// Asserts that two ULINTs are equal. If they are not, an assertion error is created.
METHOD PUBLIC AssertEquals_ULINT
VAR_INPUT
    Expected : ULINT; // ULINT expected value
    Actual : ULINT; // ULINT actual value
    Message : T_MaxString; // The identifying message for the assertion error
END_VAR
VAR
    TestInstancePath : T_MaxString;
    AlreadyReported : BOOL;
END_VAR
IF GVL_TcUnit.IgnoreCurrentTest OR GVL_TcUnit.CurrentTestIsFinished THEN
    RETURN;
END_IF

TestInstancePath := AddTestNameToInstancePath(TestInstancePath := FindTestSuiteInstancePath());

AssertResults.ReportResult(ExpectedSize := SIZEOF(Expected),
                           ExpectedTypeClass := IBaseLibrary.TypeClass.TYPE_ULINT,
                           ExpectedValue := ADR(Expected),
                           ActualSize := SIZEOF(Actual),
                           ActualTypeClass := IBaseLibrary.TypeClass.TYPE_ULINT,
                           ActualValue := ADR(Actual),
                           Message := Message,
                           TestInstancePath := TestInstancePath,
                           AlreadyReported => AlreadyReported);

IF NOT AlreadyReported AND Expected <> Actual THEN
    SetTestFailed(AssertionType := E_AssertionType.Type_ULINT,
                  AssertionMessage := Message);

    AssertMessageFormatter.LogAssertFailure(Expected := ULINT_TO_STRING(Expected),
                                            Actual := ULINT_TO_STRING(Actual),
                                            Message := Message,
                                            TestInstancePath := TestInstancePath);
END_IF
END_METHOD

// Asserts that two USINTs are equal. If they are not, an assertion error is created.
METHOD PUBLIC AssertEquals_USINT
VAR_INPUT
    Expected : USINT; // USINT expected value
    Actual : USINT; // USINT actual value
    Message : T_MaxString; // The identifying message for the assertion error
END_VAR
VAR
    AlreadyReported : BOOL;
    TestInstancePath : T_MaxString;
END_VAR
IF GVL_TcUnit.IgnoreCurrentTest OR GVL_TcUnit.CurrentTestIsFinished THEN
    RETURN;
END_IF

TestInstancePath := AddTestNameToInstancePath(TestInstancePath := FindTestSuiteInstancePath());

AssertResults.ReportResult(ExpectedSize := SIZEOF(Expected),
                           ExpectedTypeClass := IBaseLibrary.TypeClass.TYPE_USINT,
                           ExpectedValue := ADR(Expected),
                           ActualSize := SIZEOF(Actual),
                           ActualTypeClass := IBaseLibrary.TypeClass.TYPE_USINT,
                           ActualValue := ADR(Actual),
                           Message := Message,
                           TestInstancePath := TestInstancePath,
                           AlreadyReported => AlreadyReported);

IF NOT AlreadyReported AND Expected <> Actual THEN
    SetTestFailed(AssertionType := E_AssertionType.Type_USINT,
                  AssertionMessage := Message);

    AssertMessageFormatter.LogAssertFailure(Expected := USINT_TO_STRING(Expected),
                                            Actual := USINT_TO_STRING(Actual),
                                            Message := Message,
                                            TestInstancePath := TestInstancePath);
END_IF
END_METHOD

// Asserts that two WORDs are equal. If they are not, an assertion error is created.
METHOD PUBLIC AssertEquals_WORD
VAR_INPUT
    Expected : WORD; // WORD expected value
    Actual : WORD; // WORD actual value
    Message : T_MaxString; // The identifying message for the assertion error
END_VAR
VAR
    TestInstancePath : T_MaxString;
    AlreadyReported : BOOL;
END_VAR
IF GVL_TcUnit.IgnoreCurrentTest OR GVL_TcUnit.CurrentTestIsFinished THEN
    RETURN;
END_IF

TestInstancePath := AddTestNameToInstancePath(TestInstancePath := FindTestSuiteInstancePath());

AssertResults.ReportResult(ExpectedSize := SIZEOF(Expected),
                           ExpectedTypeClass := IBaseLibrary.TypeClass.TYPE_WORD,
                           ExpectedValue := ADR(Expected),
                           ActualSize := SIZEOF(Actual),
                           ActualTypeClass := IBaseLibrary.TypeClass.TYPE_WORD,
                           ActualValue := ADR(Actual),
                           Message := Message,
                           TestInstancePath := TestInstancePath,
                           AlreadyReported => AlreadyReported);

IF NOT AlreadyReported AND Expected <> Actual THEN
    SetTestFailed(AssertionType := E_AssertionType.Type_WORD,
                  AssertionMessage := Message);

    AssertMessageFormatter.LogAssertFailure(Expected := CONCAT(
                                                            STR1 := '0x',
                                                            STR2 := WORD_TO_HEXSTR(in := Expected,
                                                                                                 iPrecision := 4,
                                                                                                 bLoCase := FALSE)),
                                            Actual := CONCAT(
                                                            STR1 := '0x',
                                                            STR2 := WORD_TO_HEXSTR(in := Actual,
                                                                                                 iPrecision := 4,
                                                                                                 bLoCase := FALSE)),
                                            Message := Message,
                                            TestInstancePath := TestInstancePath);
END_IF
END_METHOD

// Asserts that two WSTRINGs are equal. If they are not, an assertion error is created.
METHOD PUBLIC AssertEquals_WSTRING
VAR_INPUT
    Expected : WSTRING(255); // WSTRING expected value
    Actual : WSTRING(255); // WSTRING actual value
    Message : T_MaxString; // The identifying message for the assertion error
END_VAR
VAR
    TestInstancePath : T_MaxString;
    AlreadyReported : BOOL;
END_VAR
IF GVL_TcUnit.IgnoreCurrentTest OR GVL_TcUnit.CurrentTestIsFinished THEN
    RETURN;
END_IF

TestInstancePath := AddTestNameToInstancePath(TestInstancePath := FindTestSuiteInstancePath());

AssertResults.ReportResult(ExpectedSize := SIZEOF(Expected),
                           ExpectedTypeClass := IBaseLibrary.TypeClass.TYPE_WSTRING,
                           ExpectedValue := ADR(Expected),
                           ActualSize := SIZEOF(Actual),
                           ActualTypeClass := IBaseLibrary.TypeClass.TYPE_WSTRING,
                           ActualValue := ADR(Actual),
                           Message := Message,
                           TestInstancePath := TestInstancePath,
                           AlreadyReported => AlreadyReported);

IF NOT AlreadyReported AND (WLEN(STR := Expected) <> WLEN(STR := Actual) OR (Expected <> Actual)) THEN
    SetTestFailed(AssertionType := E_AssertionType.Type_WSTRING,
                  AssertionMessage := Message);

    AssertMessageFormatter.LogAssertFailure(Expected := 'Not possible to print EXP unicode WSTRING value',
                                            Actual := 'Not possible to print ACT unicode WSTRING value',
                                            Message := Message,
                                            TestInstancePath := TestInstancePath);
END_IF
END_METHOD

// Asserts that a condition is false. If it is not, an assertion error is created.
METHOD PUBLIC AssertFalse
VAR_INPUT
    Condition : BOOL; // Condition to be checked
    Message : T_MaxString; // The identifying message for the assertion error
END_VAR
AssertEquals_BOOL(Expected := FALSE,
                  Actual := Condition,
                  Message := Message);
END_METHOD

// Asserts that a condition is true. If it is not, an assertion error is created.
METHOD PUBLIC AssertTrue
VAR_INPUT
    Condition : BOOL; // Condition to be checked
    Message : T_MaxString; // The identifying message for the assertion error
END_VAR
AssertEquals_BOOL(Expected := TRUE,
                  Actual := Condition,
                  Message := Message);
END_METHOD

METHOD INTERNAL CalculateAndSetNumberOfAssertsForTest
VAR_INPUT
    TestName : T_MaxString;
END_VAR
VAR
    TestInstancePath : T_MaxString;
    TotalNumberOfAsserts : UINT;
    NumberOfAsserts : UINT;
    NumberOfArrayAsserts : UINT;
    
    IteratorCounter : UINT;
END_VAR
TestInstancePath := AddTestNameToInstancePath(FindTestSuiteInstancePath());
NumberOfAsserts := AssertResults.GetNumberOfAssertsForTest(CompleteTestInstancePath := TestInstancePath);
NumberOfArrayAsserts := AssertArrayResults.GetNumberOfArrayAssertsForTest(CompleteTestInstancePath := TestInstancePath);
TotalNumberOfAsserts := NumberOfAsserts + NumberOfArrayAsserts;

IF TotalNumberOfAsserts > 0 THEN
    IF NumberOfTests > 0 THEN
        FOR IteratorCounter := 1 TO NumberOfTests BY 1 DO
            IF Tests[IteratorCounter].GetName() = TestName THEN
                Tests[IteratorCounter].SetNumberOfAssertions(NoOfAssertions := TotalNumberOfAsserts);
                RETURN;
            END_IF
        END_FOR
    END_IF
END_IF
END_METHOD

METHOD INTERNAL CalculateDuration
VAR_INPUT
    FinishedAt : LWORD; // CPU cycle counter with 100ns precision
END_VAR
IF Duration = 0.0 THEN
	Duration := LWORD_TO_LREAL(FinishedAt - StartedAt) * GVL_TcUnit.HundredNanosecondToSecond; // Seconds
	TraceWithSeverity(
		Message := CONCAT(CONCAT('SUITE COMPLETE: ', InstancePath),
				   CONCAT(' - ', CONCAT(UINT_TO_STRING(GetNumberOfSuccessfulTests()), CONCAT(' passed, ',
				   CONCAT(UINT_TO_STRING(GetNumberOfFailedTests()), CONCAT(' failed, ',
				   CONCAT(UINT_TO_STRING(GetNumberOfSkippedTests()), CONCAT(' skipped (',
				   CONCAT(LREAL_TO_STRING(Duration), 's)'))))))))),
		Severity := Global.TcEventSeverity.Info);
END_IF
END_METHOD

METHOD FB_init : BOOL
VAR_INPUT
    bInitRetains : BOOL; // if TRUE, the retain variables are initialized (warm start / cold start)
    bInCopyCode : BOOL;  // if TRUE, the instance afterwards gets moved into the copy code (online change)
END_VAR
GVL_TcUnit.NumberOfInitializedTestSuites := GVL_TcUnit.NumberOfInitializedTestSuites + 1;
GVL_TcUnit.TestSuiteAddresses[GVL_TcUnit.NumberOfInitializedTestSuites] := THIS;
END_METHOD

// Searches for the instance path of the calling function block
METHOD PRIVATE FindTestSuiteInstancePath : T_MaxString
FindTestSuiteInstancePath := GetInstancePath();
END_METHOD

METHOD INTERNAL GetDuration : LREAL
GetDuration := Duration;
END_METHOD

METHOD INTERNAL GetHasStartedRunning : BOOL
GetHasStartedRunning := StartedAt > 0;
END_METHOD

METHOD INTERNAL GetInstancePath : T_MaxString
GetInstancePath := InstancePath;
END_METHOD

METHOD INTERNAL GetNumberOfFailedTests : UINT
VAR
    Counter : UINT;
    FailedTestsCount : UINT;
    NumberOfTestsToAnalyse : UINT(1..GVL_Param_TcUnit.MaxNumberOfTestsForEachTestSuite);
    NumberOfTestOverArrayLimit : UINT;
END_VAR
// Limit the test analyse to the max array limit of 'Tests[]'
NumberOfTestsToAnalyse := GetNumberOfTestsToAnalyse();
IF GetNumberOfTests() > NumberOfTestsToAnalyse THEN
    NumberOfTestOverArrayLimit := GetNumberOfTests()-NumberOfTestsToAnalyse;
END_IF

FOR Counter := 1 TO NumberOfTestsToAnalyse BY 1 DO
    IF Tests[Counter].IsFailed() THEN
        FailedTestsCount := FailedTestsCount + 1;
    END_IF
END_FOR

GetNumberOfFailedTests := FailedTestsCount + NumberOfTestOverArrayLimit;
END_METHOD

METHOD INTERNAL GetNumberOfSkippedTests : UINT
VAR
    Counter : UINT;
    SkippedTestsCount : UINT;
    NumberOfTestsToAnalyse : UINT(1..GVL_Param_TcUnit.MaxNumberOfTestsForEachTestSuite);
END_VAR
// Limit the test analyse to the max array limit of 'Tests[]'
NumberOfTestsToAnalyse := GetNumberOfTestsToAnalyse();

FOR Counter := 1 TO NumberOfTestsToAnalyse BY 1 DO
    IF Tests[Counter].IsSkipped() THEN
        SkippedTestsCount := SkippedTestsCount + 1;
    END_IF
END_FOR

GetNumberOfSkippedTests := SkippedTestsCount;
END_METHOD

METHOD INTERNAL GetNumberOfSuccessfulTests : UINT
GetNumberOfSuccessfulTests := GetNumberOfTests() - GetNumberOfFailedTests() - GetNumberOfSkippedTests();
END_METHOD

METHOD INTERNAL GetNumberOfTests : UINT
GetNumberOfTests := NumberOfTests;
END_METHOD

METHOD INTERNAL GetNumberOfTestsToAnalyse : UINT
GetNumberOfTestsToAnalyse := MIN(GetNumberOfTests(), GVL_Param_TcUnit.MaxNumberOfTestsForEachTestSuite);
END_METHOD

METHOD GetTestByName : REFERENCE TO FB_Test
VAR_INPUT
  TestName : T_MaxString;
END_VAR
VAR
  IteratorCounter : UINT;
  NumberOfTestsToAnalyse : UINT(1..GVL_Param_TcUnit.MaxNumberOfTestSuites);
END_VAR
NumberOfTestsToAnalyse := GetNumberOfTestsToAnalyse();
FOR IteratorCounter := 1 TO NumberOfTestsToAnalyse BY 1 DO
  IF Tests[IteratorCounter].GetName() = TestName THEN
    GetTestByName REF= Tests[IteratorCounter];
    RETURN;
	END_IF
END_FOR
END_METHOD

// This method returns the test at the n'th position, ranging from 1.. NumberOfTests
METHOD INTERNAL GetTestByPosition : FB_Test
VAR_INPUT
    Position : UINT(1..GVL_Param_TcUnit.MaxNumberOfTestsForEachTestSuite);
END_VAR
GetTestByPosition := Tests[Position];
END_METHOD

METHOD INTERNAL GetTestOrderNumber : UINT(0..GVL_Param_TcUnit.MaxNumberOfTestsForEachTestSuite);
VAR_INPUT
    TestName : T_MaxString;
END_VAR
VAR
    IteratorCounter : UINT;
    NumberOfTestsToAnalyse : UINT(1..GVL_Param_TcUnit.MaxNumberOfTestsForEachTestSuite);
END_VAR
// Limit the test analyse to the max array limit of 'Tests[]'
NumberOfTestsToAnalyse := GetNumberOfTestsToAnalyse();

FOR IteratorCounter := 1 TO NumberOfTestsToAnalyse BY 1 DO
    IF Tests[IteratorCounter].GetName() = TestName THEN
        GetTestOrderNumber := Tests[IteratorCounter].GetTestOrder();
        RETURN;
    END_IF
END_FOR
END_METHOD

METHOD INTERNAL IsTestFinished : BOOL
VAR_INPUT
    TestName : T_MaxString;
END_VAR
VAR
    IteratorCounter : UINT;
    NumberOfTestsToAnalyse : UINT(0..GVL_Param_TcUnit.MaxNumberOfTestsForEachTestSuite);
END_VAR
// Limit the test analyse to the max array limit of 'Tests[]'
NumberOfTestsToAnalyse := GetNumberOfTestsToAnalyse();

IsTestFinished := FALSE;
FOR IteratorCounter := 1 TO NumberOfTestsToAnalyse BY 1 DO
    IF Tests[IteratorCounter].GetName() = TestName THEN
        IsTestFinished := Tests[IteratorCounter].IsFinished();
        RETURN;
    END_IF
END_FOR
END_METHOD

METHOD INTERNAL SetStartedAtIfNotSet
VAR_INPUT
    Timestamp : LWORD; // CPU cycle counter with 100ns precision
END_VAR
IF StartedAt = 0 THEN
    StartedAt := Timestamp;
END_IF
END_METHOD

METHOD INTERNAL SetStartedAtTimeBasedOnCpuCounter
StartedAt := F_GetCpuCounterAs64bit(GVL_TcUnit.GetCpuCounter);
END_METHOD

METHOD INTERNAL SetTestFailed
VAR_INPUT
    AssertionType : E_AssertionType;
    AssertionMessage : T_MaxString;
END_VAR
VAR
    IteratorCounter : UINT;
    NumberOfTestsToAnalyse : UINT(0..GVL_Param_TcUnit.MaxNumberOfTestsForEachTestSuite);
END_VAR
// Limit the test analyse to the max array limit of 'Tests[]'
NumberOfTestsToAnalyse := GetNumberOfTestsToAnalyse();

FOR IteratorCounter := 1 TO NumberOfTestsToAnalyse BY 1 DO
    IF Tests[IteratorCounter].GetName() = GVL_TcUnit.CurrentTestNameBeingCalled THEN
        Tests[IteratorCounter].SetFailed();
        Tests[IteratorCounter].SetAssertionType(AssertType := AssertionType);
        Tests[IteratorCounter].SetAssertionMessage(AssertMessage := AssertionMessage);
    END_IF
END_FOR
END_METHOD

(* Marks the test as finished in this testsuite.
   Returns TRUE if test was found, and FALSE if a test with this name was not found in this testsuite *)
METHOD INTERNAL SetTestFinished : BOOL;
VAR_INPUT
    TestName : T_MaxString;
    FinishedAt : LWORD;
END_VAR
VAR
    IteratorCounter : UINT;
    NumberOfTestsToAnalyse : UINT(0..GVL_Param_TcUnit.MaxNumberOfTestsForEachTestSuite);
END_VAR
// Limit the test analyse to the max array limit of 'Tests[]'
NumberOfTestsToAnalyse := GetNumberOfTestsToAnalyse();
FOR IteratorCounter := 1 TO NumberOfTestsToAnalyse BY 1 DO
    IF Tests[IteratorCounter].GetName() = TestName THEN
		IF NOT Tests[IteratorCounter].IsFinished() THEN
        	Tests[IteratorCounter].SetFinishedAndDuration(FinishedAt := FinishedAt);
			IF Tests[IteratorCounter].IsFailed() THEN
				TraceWithSeverity(
					Message := CONCAT(CONCAT('TEST FAILED: ', TestName),
							   CONCAT(' (', CONCAT(LREAL_TO_STRING(Tests[IteratorCounter].GetDuration()), 's)'))),
					Severity := Global.TcEventSeverity.Warning);
			ELSE
				TraceWithSeverity(
					Message := CONCAT(CONCAT('TEST PASSED: ', TestName),
							   CONCAT(' (', CONCAT(LREAL_TO_STRING(Tests[IteratorCounter].GetDuration()), 's)'))),
					Severity := Global.TcEventSeverity.Info);
			END_IF
		END_IF
		SetTestFinished := TRUE;
        RETURN;
    END_IF
END_FOR
SetTestFinished := FALSE;
END_METHOD

END_FUNCTION_BLOCK

// POUs/FB_xUnitXmlPublisher
// Publishes test results into an xUnit compatible Xml file
FUNCTION_BLOCK FB_xUnitXmlPublisher EXTENDS FB_BaseStatic IMPLEMENTS I_TestResultLogger
VAR
    // Dependency injection via FB_Init
    TestResults : I_TestResults;

    // File access mode
    AccessMode : SysFile.ACCESS_MODE := SysFile.AM_WRITE_PLUS;

    File : FB_FileControl;
    Xml : FB_XMLControl;
    BufferInitialised : BOOL := FALSE;
    Buffer : ARRAY [0..(GVL_Param_TcUnit.XUnitBufferSize - 1)] OF BYTE;
    WritingTestSuiteResultNumber : UINT(1..GVL_Param_TcUnit.MaxNumberOfTestSuites);
    PublishTrigger : R_TRIG;
END_VAR

(*
    Deletes the former file (if it exists).
    Opens the file, writes the buffer and closes it.
*)
METHOD PRIVATE DeleteOpenWriteClose : SysFile.SysTypes.RTS_IEC_RESULT;
VAR
    WriteResult : SysFile.SysTypes.RTS_IEC_RESULT;
END_VAR
DeleteOpenWriteClose := SysDir.CmpErrors.Errors.ERR_OK;
IF Initialised() THEN
    // Delete may fail if file doesn't exist yet (first run) — not a real error
    DeleteOpenWriteClose := MAX(DeleteOpenWriteClose, File.Delete(Filename := GVL_Param_TcUnit.xUnitFilePath));
    // Track Open/Write/Close separately for trace — these are the real errors
    WriteResult := File.Open(Filename := GVL_Param_TcUnit.xUnitFilePath, FileAccessMode := AccessMode);
    WriteResult := MAX(WriteResult, File.Write(BufferPointer := ADR(Buffer), Xml.Length));
    WriteResult := MAX(WriteResult, File.Close());
    DeleteOpenWriteClose := MAX(DeleteOpenWriteClose, WriteResult);
ELSE
    WriteResult := SysDir.CmpErrors.Errors.ERR_NOBUFFER;
    DeleteOpenWriteClose := WriteResult;
END_IF;

IF WriteResult <> SysDir.CmpErrors.Errors.ERR_OK THEN
    TraceWithSeverity(
        Message := CONCAT('xUnit file I/O failure: ', GVL_Param_TcUnit.xUnitFilePath),
        Severity := Global.TcEventSeverity.Error);
END_IF;
END_METHOD

(*
    FB_Init is always available implicitly AND it is used primarily FOR initialization.
    The return value is not evaluated. For a specific influence, you can also declare the
    methods explicitly and provide additional code there with the standard initialization
    code. You can evaluate the return value.
*)
METHOD FB_Init: BOOL
VAR_INPUT
    bInitRetains: BOOL; // TRUE: the retain variables are initialized (reset warm / reset cold)
    bInCopyCode: BOOL;  // TRUE: the instance will be copied to the copy code afterward (online change)
    iTestResults : I_TestResults; // Interface dependency injection
END_VAR
// Set buffer and flag
Xml.SetBuffer(PointerToBuffer := ADR(Buffer), SizeOfBuffer := SIZEOF(Buffer));

// Set buffer initialised
BufferInitialised := TRUE;

// Set testresult interface
THIS^.TestResults := iTestResults;
END_METHOD

METHOD PRIVATE Initialised : BOOL
Initialised := THIS^.BufferInitialised;
END_METHOD

(*
    This method is responsible for the entire generation of the output file. 
    The output of the xml writer is NOT beautified.

    When new data is available, feel free to add it to the report
*)
METHOD PUBLIC LogTestSuiteResults
VAR
    UnitTestResults : REFERENCE TO ST_TestSuiteResults;
    CurrentSuiteNumber : UINT;
    CurrentTestCount : UINT;
END_VAR
VAR CONSTANT
    TEST_STATUS_SKIP : STRING := 'SKIP';
    TEST_STATUS_PASS : STRING := 'PASS';
    TEST_STATUS_FAIL : STRING := 'FAIL';
END_VAR
UnitTestResults REF= TestResults.GetTestSuiteResults();

// Only publish once if "GVL_Param_TcUnit.xUnitEnablePublish" is enabled and all test results are stored.
PublishTrigger(CLK := (TestResults.GetAreTestResultsAvailable() AND GVL_Param_TcUnit.xUnitEnablePublish));
IF PublishTrigger.Q THEN

    // <?xml version="1.0" encoding="UTF-8"?>
    Xml.WriteDocumentHeader(Header := '<?xml version="1.0" encoding="UTF-8"?>');

    // <testsuites>  ('disabled' removed 2026-07-18: an empty string breaks JUnit
    //  parsers expecting an integer; skipped counts carry the information)
    Xml.NewTag('testsuites');
    Xml.NewParameter('failures', UDINT_TO_STRING(UnitTestResults.NumberOfFailedTestCases));
    (* 'tests' is the TOTAL testcase count; the previous successful-only value was a bug *)
    Xml.NewParameter('tests', UDINT_TO_STRING(UnitTestResults.NumberOfTestCases));
    Xml.NewParameter('skipped', UDINT_TO_STRING(UnitTestResults.NumberOfSkippedTestCases));
    Xml.NewParameter('time', LREAL_TO_STRING(UnitTestResults.Duration));

    FOR CurrentSuiteNumber := 1 TO UnitTestResults.NumberOfTestSuites BY 1 DO
        // <testsuite>
        Xml.NewTag('testsuite');
        Xml.NewParameter('id', UINT_TO_STRING(UnitTestResults.TestSuiteResults[CurrentSuiteNumber].Identity));
        Xml.NewParameter('name', UnitTestResults.TestSuiteResults[CurrentSuiteNumber].name);
        Xml.NewParameter('tests', UINT_TO_STRING(UnitTestResults.TestSuiteResults[CurrentSuiteNumber].NumberOfTests));
        Xml.NewParameter('failures', UINT_TO_STRING(UnitTestResults.TestSuiteResults[CurrentSuiteNumber].NumberOfFailedTests));
        Xml.NewParameter('skipped', UINT_TO_STRING(UnitTestResults.TestSuiteResults[CurrentSuiteNumber].NumberOfSkippedTests));
        Xml.NewParameter('time', LREAL_TO_STRING(UnitTestResults.TestSuiteResults[CurrentSuiteNumber].Duration));

        FOR CurrentTestCount := 1 TO UnitTestResults.TestSuiteResults[CurrentSuiteNumber].NumberOfTests BY 1 DO
            // <testcase>
            Xml.NewTag('testcase');
            Xml.NewParameter('name', UnitTestResults.TestSuiteResults[CurrentSuiteNumber].TestCaseResults[CurrentTestCount].TestName);
            Xml.NewParameter('classname', UnitTestResults.TestSuiteResults[CurrentSuiteNumber].TestCaseResults[CurrentTestCount].TestClassName);
            Xml.NewParameter('time', LREAL_TO_STRING(UnitTestResults.TestSuiteResults[CurrentSuiteNumber].TestCaseResults[CurrentTestCount].Duration));

            IF UnitTestResults.TestSuiteResults[CurrentSuiteNumber].TestCaseResults[CurrentTestCount].TestIsFailed THEN
                Xml.NewParameter('status', TEST_STATUS_FAIL);
            ELSIF UnitTestResults.TestSuiteResults[CurrentSuiteNumber].TestCaseResults[CurrentTestCount].TestIsSkipped THEN
                Xml.NewParameter('status', TEST_STATUS_SKIP);
            ELSE
                Xml.NewParameter('status', TEST_STATUS_PASS);
            END_IF

            // Determine testcase fail, skip, or success
            IF UnitTestResults.TestSuiteResults[CurrentSuiteNumber].TestCaseResults[CurrentTestCount].FailureType <> E_AssertionType.Type_UNDEFINED THEN
                (* In case of fail
                    <failure message="Values differ" type="BYTE" />
                *)
                Xml.NewTag('failure');
                Xml.NewParameter('message', UnitTestResults.TestSuiteResults[CurrentSuiteNumber].TestCaseResults[CurrentTestCount].FailureMessage);
                Xml.NewParameter('type', F_AssertionTypeToString(UnitTestResults.TestSuiteResults[CurrentSuiteNumber].TestCaseResults[CurrentTestCount].FailureType));
                // Close failure tag
                Xml.CloseTag();
            ELSIF UnitTestResults.TestSuiteResults[CurrentSuiteNumber].TestCaseResults[CurrentTestCount].TestIsSkipped THEN
                (* JUnit consumers recognize a skipped testcase through a <skipped/>
                   child element, not a custom status attribute (kept for
                   backward compatibility) *)
                Xml.NewTag('skipped');
                Xml.CloseTag();
            ELSE
            // In case of success
            Xml.NewTagData('');

            END_IF
            // Close testcase tag
            Xml.CloseTag();

        END_FOR
        // Close testsuite tag
        Xml.CloseTag();

    END_FOR
    // Close testsuites
    Xml.CloseTag();

    // Delete, open, save and close the file
    DeleteOpenWriteClose();

    // Clear the internal buffer
    Xml.ClearBuffer();

    // Inform user
    GVL_TcUnit.AdsMessageQueue.WriteLog(MsgCtrlMask := ADSLOG_MSGTYPE_HINT,
                                        msgFmtStr := '%s',
                                        strArg := '| ==========TEST RESULTS EXPORTED===========');

    GVL_TcUnit.AdsMessageQueue.WriteLog(MsgCtrlMask := ADSLOG_MSGTYPE_HINT,
                                        msgFmtStr :=  '| Location: %s ',
                                        strArg := GVL_Param_TcUnit.xUnitFilePath);

    GVL_TcUnit.AdsMessageQueue.WriteLog(MsgCtrlMask := ADSLOG_MSGTYPE_HINT,
                                        MsgFmtStr := '%s',
                                        StrArg := '| ======================================');

    TraceWithSeverity(
        Message := CONCAT('xUnit XML exported to ', GVL_Param_TcUnit.xUnitFilePath),
        Severity := Global.TcEventSeverity.Info);
END_IF
END_METHOD

END_FUNCTION_BLOCK

// POUs/FB_TimedTestSuite
FUNCTION_BLOCK FB_TimedTestSuite EXTENDS FB_TestSuite
VAR
    TimedTestStates      : ARRAY[1..GVL_Param_TcUnit.MaxNumberOfTestsForEachTestSuite] OF ST_TimedTestState;
    _nActiveTimedTestIdx : UINT;
    (* Task cycle in which _nActiveTimedTestIdx was set; a wait helper only accepts
       the context if it was set in the same cycle (guards cross-scan staleness) *)
    _nActiveTimedTestCycle : UDINT;
    // One-shot for the out-of-context wait Error trace (cyclic path - must not storm)
    bOutOfContextWaitTraced : BOOL;
END_VAR

METHOD PRIVATE _FindTestIndex : UINT
VAR_INPUT
    TestName : T_MaxString;
END_VAR
VAR
    i : UINT;
    nMax : UINT;
END_VAR
_FindTestIndex := 0;
nMax := GetNumberOfTestsToAnalyse();
FOR i := 1 TO nMax BY 1 DO
    IF Tests[i].GetName() = TestName THEN
        _FindTestIndex := i;
        RETURN;
    END_IF
END_FOR
END_METHOD

(* Returns the timed-test index for a wait-helper call, or 0 when the call is
   out of context. Valid context requires all three: an index was set, it was
   set in the current task cycle (TEST_TIMED* ran earlier in this scan and
   selected this test for body execution), and the framework's current test
   name still matches (defense against later TEST() calls in the same scan). *)
METHOD PRIVATE _GetActiveWaitContext : UINT
VAR
    idx : UINT;
END_VAR
_GetActiveWaitContext := 0;
idx := _nActiveTimedTestIdx;
IF idx = 0 THEN
    RETURN;
END_IF

GetCurrentTaskIndex();
IF _nActiveTimedTestCycle <> TwinCAT_SystemInfoVarList._TaskInfo[GetCurrentTaskIndex.index].CycleCount THEN
    RETURN;
END_IF

IF Tests[idx].GetName() <> GVL_TcUnit.CurrentTestNameBeingCalled THEN
    RETURN;
END_IF

_GetActiveWaitContext := idx;
END_METHOD

METHOD PUBLIC GetTimedTestResult : ST_TimedTestResult
VAR_INPUT
    TestName : T_MaxString;
END_VAR
VAR
    idx  : UINT;
    Test : REFERENCE TO FB_Test;
END_VAR
// Normalize the same way TEST(), TEST_ORDERED(), and TEST_TIMED() do
TestName := F_LTrim(in := F_RTrim(in := TestName));

idx := _FindTestIndex(TestName := TestName);
IF idx = 0 THEN
    RETURN;
END_IF

Test REF= Tests[idx];
IF NOT __ISVALIDREF(Test) THEN
    RETURN;
END_IF

GetTimedTestResult.TestName := Test.GetName();
GetTimedTestResult.bIsFailed := Test.IsFailed();
GetTimedTestResult.bIsSkipped := Test.IsSkipped();
GetTimedTestResult.bIsFinished := Test.IsFinished();
GetTimedTestResult.sFailureMessage := Test.GetAssertionMessage();
GetTimedTestResult.eFailureType := Test.GetAssertionType();
GetTimedTestResult.nNumberOfAsserts := Test.GetNumberOfAssertions();
GetTimedTestResult.lrDuration := Test.GetDuration();
GetTimedTestResult.stTimedState := TimedTestStates[idx];
END_METHOD

METHOD PUBLIC TEST_TIMED : BOOL
VAR_INPUT
    TestName       : T_MaxString;
    tSafetyTimeout : TIME;
END_VAR
VAR
    idx         : UINT;
    lrElapsed   : LREAL;
    lrTimeout   : LREAL;
    sMsg        : T_MaxString;
END_VAR
TEST_TIMED := FALSE;

// Step 1: Reset context
_nActiveTimedTestIdx := 0;

// Step 2: Trim name
TestName := F_LTrim(in := F_RTrim(in := TestName));

// Step 3: Register test via free function TEST()
TEST(TestName := TestName);

// Step 4: Check skip/ignore
IF GVL_TcUnit.IgnoreCurrentTest THEN
    RETURN;
END_IF

// Step 5: Find test index
idx := _FindTestIndex(TestName := TestName);
IF idx = 0 THEN
    RETURN;
END_IF

// Step 6: Check already finished
IF TimedTestStates[idx].bSafetyTimedOut OR IsTestFinished(TestName := TestName) THEN
    GVL_TcUnit.CurrentTestIsFinished := TRUE;
    RETURN;
END_IF

// Step 7: Initialize on first call
IF NOT TimedTestStates[idx].bInitialized THEN
    TimedTestStates[idx].nSafetyStartTime := F_GetCpuCounterAs64bit(GVL_TcUnit.GetCpuCounter);
    TimedTestStates[idx].tSafetyTimeout := tSafetyTimeout;
    TimedTestStates[idx].bInitialized := TRUE;
END_IF

// Step 8: Check safety timeout (compare against stored value)
lrElapsed := ULINT_TO_LREAL(F_GetCpuCounterAs64bit(GVL_TcUnit.GetCpuCounter) - TimedTestStates[idx].nSafetyStartTime)
             * GVL_TcUnit.HundredNanosecondToSecond;
lrTimeout := TIME_TO_LREAL(TimedTestStates[idx].tSafetyTimeout) / 1000.0;

IF lrElapsed > lrTimeout THEN
    sMsg := CONCAT('SAFETY TIMEOUT: Test "', CONCAT(TestName, CONCAT('" exceeded ', LREAL_TO_FMTSTR(lrTimeout, 1, TRUE))));
    sMsg := CONCAT(sMsg, 's');

    SetTestFailed(AssertionType := E_AssertionType.Type_TIMEOUT,
                  AssertionMessage := sMsg);
    SetTestFinished(TestName := TestName,
                    FinishedAt := F_GetCpuCounterAs64bit(GVL_TcUnit.GetCpuCounter));
    CalculateAndSetNumberOfAssertsForTest(TestName := TestName);

    TimedTestStates[idx].bSafetyTimedOut := TRUE;
    GVL_TcUnit.CurrentTestIsFinished := TRUE;

    TraceWithSeverity(Message := sMsg, Severity := TcEventSeverity.Warning);
    RETURN;
END_IF

// Step 9: Test body should execute - arm the wait context for this cycle only
_nActiveTimedTestIdx := idx;
GetCurrentTaskIndex();
_nActiveTimedTestCycle := TwinCAT_SystemInfoVarList._TaskInfo[GetCurrentTaskIndex.index].CycleCount;
TEST_TIMED := TRUE;
END_METHOD

METHOD PUBLIC TEST_TIMED_ORDERED : BOOL
VAR_INPUT
    TestName       : T_MaxString;
    tSafetyTimeout : TIME;
END_VAR
VAR
    CounterTestSuiteAddress : UINT;
    SuiteIndex              : UINT;
    Test                    : REFERENCE TO FB_Test;
    idx                     : UINT;
    lrElapsed               : LREAL;
    lrTimeout               : LREAL;
    sMsg                    : T_MaxString;
END_VAR
TEST_TIMED_ORDERED := FALSE;

// Step 1: Reset context
_nActiveTimedTestIdx := 0;

// Step 2: Trim name (matches TEST_ORDERED line 34)
TestName := F_LTrim(in := F_RTrim(in := TestName));

// Step 3: Set global test name (matches line 37)
GVL_TcUnit.CurrentTestNameBeingCalled := TestName;

// Step 4: Find suite in runner registry (matches lines 44-47)
SuiteIndex := 0;
FOR CounterTestSuiteAddress := 1 TO GVL_TcUnit.NumberOfInitializedTestSuites BY 1 DO
    IF GVL_TcUnit.TestSuiteAddresses[CounterTestSuiteAddress] = GVL_TcUnit.CurrentTestSuiteBeingCalled THEN
        SuiteIndex := CounterTestSuiteAddress;
        EXIT;
    END_IF
END_FOR
IF SuiteIndex = 0 THEN
    RETURN;
END_IF

// Step 5: Register as ordered test (matches line 48)
Test REF= GVL_TcUnit.TestSuiteAddresses[SuiteIndex]^.AddTest(TestName := TestName, IsTestOrdered := TRUE);

// Step 6: Set CurrentTestIsFinished (matches line 49)
GVL_TcUnit.CurrentTestIsFinished := GVL_TcUnit.TestSuiteAddresses[SuiteIndex]^.IsTestFinished(TestName := TestName);

// Step 7: Check skip/ignore (matches lines 76-78)
IF GVL_TcUnit.IgnoreCurrentTest THEN
    RETURN;
END_IF

// Step 8: Check ordered cursor (matches lines 55-74)
IF GetTestOrderNumber(TestName := TestName) = GVL_TcUnit.CurrentlyRunningOrderedTestInTestSuite[SuiteIndex] THEN
    IF GVL_TcUnit.CurrentTestIsFinished THEN
        // Already finished - advance cursor (matches lines 58-62)
        GVL_TcUnit.CurrentlyRunningOrderedTestInTestSuite[SuiteIndex] :=
            GVL_TcUnit.CurrentlyRunningOrderedTestInTestSuite[SuiteIndex] + 1;
        GVL_TcUnit.IgnoreCurrentTest := TRUE;
        RETURN;
    END_IF
ELSE
    // Not this test's turn (matches lines 70-73)
    GVL_TcUnit.IgnoreCurrentTest := TRUE;
    RETURN;
END_IF

// --- From here: this test's turn AND not finished. Add timed-test logic. ---

// Step 9: Find timed test index
idx := _FindTestIndex(TestName := TestName);
IF idx = 0 THEN
    RETURN;
END_IF

// Step 10: Check already timed out
IF TimedTestStates[idx].bSafetyTimedOut THEN
    GVL_TcUnit.CurrentTestIsFinished := TRUE;
    RETURN;
END_IF

// Step 11: Initialize on first call
IF NOT TimedTestStates[idx].bInitialized THEN
    TimedTestStates[idx].nSafetyStartTime := F_GetCpuCounterAs64bit(GVL_TcUnit.GetCpuCounter);
    TimedTestStates[idx].tSafetyTimeout := tSafetyTimeout;
    TimedTestStates[idx].bInitialized := TRUE;
END_IF

// Step 12: Check safety timeout (compare against stored value)
lrElapsed := ULINT_TO_LREAL(F_GetCpuCounterAs64bit(GVL_TcUnit.GetCpuCounter) - TimedTestStates[idx].nSafetyStartTime)
             * GVL_TcUnit.HundredNanosecondToSecond;
lrTimeout := TIME_TO_LREAL(TimedTestStates[idx].tSafetyTimeout) / 1000.0;

IF lrElapsed > lrTimeout THEN
    sMsg := CONCAT('SAFETY TIMEOUT: Test "', CONCAT(TestName, CONCAT('" exceeded ', LREAL_TO_FMTSTR(lrTimeout, 1, TRUE))));
    sMsg := CONCAT(sMsg, 's');

    SetTestFailed(AssertionType := E_AssertionType.Type_TIMEOUT,
                  AssertionMessage := sMsg);
    SetTestFinished(TestName := TestName,
                    FinishedAt := F_GetCpuCounterAs64bit(GVL_TcUnit.GetCpuCounter));
    CalculateAndSetNumberOfAssertsForTest(TestName := TestName);

    TimedTestStates[idx].bSafetyTimedOut := TRUE;
    GVL_TcUnit.CurrentTestIsFinished := TRUE;

    TraceWithSeverity(Message := sMsg, Severity := TcEventSeverity.Warning);
    RETURN;
END_IF

// Step 13: Set started timestamp (matches line 66)
IF __ISVALIDREF(Test) THEN
    Test.SetStartedAtIfNotSet(Timestamp := F_GetCpuCounterAs64bit(GVL_TcUnit.GetCpuCounter));
END_IF

// Step 14: Test body should execute - arm the wait context for this cycle only
_nActiveTimedTestIdx := idx;
GetCurrentTaskIndex();
_nActiveTimedTestCycle := TwinCAT_SystemInfoVarList._TaskInfo[GetCurrentTaskIndex.index].CycleCount;
TEST_TIMED_ORDERED := TRUE;
END_METHOD

METHOD PUBLIC WaitForCondition : BOOL
VAR_INPUT
    bCondition : BOOL;
    tTimeout   : TIME;
END_VAR
VAR
    idx       : UINT;
    lrElapsed : LREAL;
    lrTarget  : LREAL;
END_VAR
WaitForCondition := FALSE;
idx := _GetActiveWaitContext();

// Step 1: Context check (one-shot trace - this path is cyclic)
IF idx = 0 THEN
    IF NOT bOutOfContextWaitTraced THEN
        bOutOfContextWaitTraced := TRUE;
        TraceWithSeverity(
            Message := 'WaitForCondition called without active timed test context',
            Severity := TcEventSeverity.Error);
    END_IF
    RETURN;
END_IF

// Step 2: Pass-through if already complete
IF TimedTestStates[idx].bWaitComplete THEN
    WaitForCondition := TRUE;
    RETURN;
END_IF

// Step 3: Type mismatch check
IF TimedTestStates[idx].eWaitType = E_WaitType.Duration THEN
    SetTestFailed(AssertionType := E_AssertionType.Type_WAIT_MISUSE,
                  AssertionMessage := 'WaitForCondition called but WaitForTime already active');
    SetTestFinished(TestName := GVL_TcUnit.CurrentTestNameBeingCalled,
                    FinishedAt := F_GetCpuCounterAs64bit(GVL_TcUnit.GetCpuCounter));
    CalculateAndSetNumberOfAssertsForTest(TestName := GVL_TcUnit.CurrentTestNameBeingCalled);
    GVL_TcUnit.CurrentTestIsFinished := TRUE;
    RETURN;
END_IF

// Step 4: First call with condition already TRUE - immediate completion
IF bCondition AND TimedTestStates[idx].nWaitStartTime = 0 THEN
    TimedTestStates[idx].bWaitComplete := TRUE;
    TimedTestStates[idx].bConditionTimedOut := FALSE;
    TimedTestStates[idx].eWaitType := E_WaitType.Condition;
    TraceWithSeverity(
        Message := CONCAT('WaitForCondition: condition already TRUE for test "', CONCAT(GVL_TcUnit.CurrentTestNameBeingCalled, '"')),
        Severity := TcEventSeverity.Info);
    WaitForCondition := TRUE;
    RETURN;
END_IF

// Step 5: First call, condition not yet met - start wait
IF TimedTestStates[idx].nWaitStartTime = 0 THEN
    TimedTestStates[idx].eWaitType := E_WaitType.Condition;
    TimedTestStates[idx].tLatchedDuration := tTimeout;
    TimedTestStates[idx].nWaitStartTime := F_GetCpuCounterAs64bit(GVL_TcUnit.GetCpuCounter);
    TraceWithSeverity(
        Message := CONCAT('WaitForCondition started: timeout ', CONCAT(TIME_TO_STRING(tTimeout), CONCAT(' for test "', CONCAT(GVL_TcUnit.CurrentTestNameBeingCalled, '"')))),
        Severity := TcEventSeverity.Verbose);
    RETURN;
END_IF

// Step 6: Condition met during wait
IF bCondition THEN
    TimedTestStates[idx].bWaitComplete := TRUE;
    TimedTestStates[idx].bConditionTimedOut := FALSE;
    TraceWithSeverity(
        Message := CONCAT('WaitForCondition: condition met for test "', CONCAT(GVL_TcUnit.CurrentTestNameBeingCalled, '"')),
        Severity := TcEventSeverity.Info);
    WaitForCondition := TRUE;
    RETURN;
END_IF

// Step 7: Check timeout
lrElapsed := ULINT_TO_LREAL(F_GetCpuCounterAs64bit(GVL_TcUnit.GetCpuCounter) - TimedTestStates[idx].nWaitStartTime)
             * GVL_TcUnit.HundredNanosecondToSecond;
lrTarget := TIME_TO_LREAL(TimedTestStates[idx].tLatchedDuration) / 1000.0;

IF lrElapsed >= lrTarget THEN
    TimedTestStates[idx].bWaitComplete := TRUE;
    TimedTestStates[idx].bConditionTimedOut := TRUE;
    TraceWithSeverity(
        Message := CONCAT('WaitForCondition timed out after ', CONCAT(LREAL_TO_FMTSTR(lrElapsed, 3, TRUE), CONCAT('s for test "', CONCAT(GVL_TcUnit.CurrentTestNameBeingCalled, '"')))),
        Severity := TcEventSeverity.Warning);
    WaitForCondition := TRUE;
END_IF

// Step 8: Still waiting - return FALSE (default)
END_METHOD

METHOD PUBLIC WaitForTime : BOOL
VAR_INPUT
    tDuration : TIME;
END_VAR
VAR
    idx       : UINT;
    lrElapsed : LREAL;
    lrTarget  : LREAL;
END_VAR
WaitForTime := FALSE;
idx := _GetActiveWaitContext();

// Step 1: Context check (one-shot trace - this path is cyclic)
IF idx = 0 THEN
    IF NOT bOutOfContextWaitTraced THEN
        bOutOfContextWaitTraced := TRUE;
        TraceWithSeverity(
            Message := 'WaitForTime called without active timed test context',
            Severity := TcEventSeverity.Error);
    END_IF
    RETURN;
END_IF

// Step 2: Pass-through if already complete
IF TimedTestStates[idx].bWaitComplete THEN
    WaitForTime := TRUE;
    RETURN;
END_IF

// Step 3: Type mismatch check
IF TimedTestStates[idx].eWaitType = E_WaitType.Condition THEN
    SetTestFailed(AssertionType := E_AssertionType.Type_WAIT_MISUSE,
                  AssertionMessage := 'WaitForTime called but WaitForCondition already active');
    SetTestFinished(TestName := GVL_TcUnit.CurrentTestNameBeingCalled,
                    FinishedAt := F_GetCpuCounterAs64bit(GVL_TcUnit.GetCpuCounter));
    CalculateAndSetNumberOfAssertsForTest(TestName := GVL_TcUnit.CurrentTestNameBeingCalled);
    GVL_TcUnit.CurrentTestIsFinished := TRUE;
    RETURN;
END_IF

// Step 4: First call - start wait
IF TimedTestStates[idx].nWaitStartTime = 0 THEN
    TimedTestStates[idx].eWaitType := E_WaitType.Duration;
    TimedTestStates[idx].tLatchedDuration := tDuration;
    TimedTestStates[idx].nWaitStartTime := F_GetCpuCounterAs64bit(GVL_TcUnit.GetCpuCounter);
    TraceWithSeverity(
        Message := CONCAT('Wait started: ', CONCAT(TIME_TO_STRING(tDuration), CONCAT(' for test "', CONCAT(GVL_TcUnit.CurrentTestNameBeingCalled, '"')))),
        Severity := TcEventSeverity.Verbose);
    RETURN;
END_IF

// Steps 5-8: Check elapsed
lrElapsed := ULINT_TO_LREAL(F_GetCpuCounterAs64bit(GVL_TcUnit.GetCpuCounter) - TimedTestStates[idx].nWaitStartTime)
             * GVL_TcUnit.HundredNanosecondToSecond;
lrTarget := TIME_TO_LREAL(TimedTestStates[idx].tLatchedDuration) / 1000.0;

IF lrElapsed >= lrTarget THEN
    TimedTestStates[idx].bWaitComplete := TRUE;
    TraceWithSeverity(
        Message := CONCAT('Wait completed: ', CONCAT(LREAL_TO_FMTSTR(lrElapsed, 3, TRUE), CONCAT('s elapsed for test "', CONCAT(GVL_TcUnit.CurrentTestNameBeingCalled, '"')))),
        Severity := TcEventSeverity.Info);
    WaitForTime := TRUE;
END_IF
END_METHOD

PROPERTY PUBLIC WaitTimedOut : BOOL
GET
VAR
    idx : UINT;
END_VAR
idx := _GetActiveWaitContext();
IF idx > 0 THEN
    WaitTimedOut := TimedTestStates[idx].bConditionTimedOut;
ELSE
    WaitTimedOut := FALSE;
END_IF
END_GET
END_PROPERTY

END_FUNCTION_BLOCK
